FUNCTION_BLOCK FB_TestableCarryoverSubStateService EXTENDS FB_ServiceBase
VAR
	// Simulate a second run that still holds the previous run's final substate.
	_Step : UDINT := 5;
END_VAR

M_UpdateService(CompletionBehavior := E_ServiceCompletionBehavior.NaturalCompletion);

METHOD PROTECTED H_GetExecuteSubState : UDINT
H_GetExecuteSubState := _Step;
END_METHOD

METHOD PROTECTED H_GetExecuteSubStateName : STRING(80)
CASE _Step OF
	1: H_GetExecuteSubStateName := 'LiftReady';
	5: H_GetExecuteSubStateName := 'Finish';
ELSE
	H_GetExecuteSubStateName := '';
END_CASE
END_METHOD

METHOD PROTECTED H_OnExecute : E_PackMLHookResult
VAR_INPUT
	bFirstScan : BOOL;
END_VAR
IF bFirstScan THEN
	_Step := 1;
END_IF
H_OnExecute := E_PackMLHookResult.Busy;
END_METHOD

END_FUNCTION_BLOCK

(* stored: Version 1.1.0.1, ProductVersion 3.1.4026.18
   POU FB_TestableCarryoverSubStateService: Id {2e98a9ae-b2b7-46bc-94c1-8fc05d7b0b5a}, SpecialFunc None
   Method H_GetExecuteSubState: Id {7feac875-9e4c-481a-87d4-dccfc80d819e}
   Method H_GetExecuteSubStateName: Id {612301a6-f8c6-4d75-8d0d-bd9f517b57f4}
   Method H_OnExecute: Id {50323b34-6b9f-432f-a631-ea17ee71161b} *)
